(* PLC project Tc2_Utilities.PLC_ReadSymInfoByName Demo, tc3-libraries-kb TwinCAT 3.1 *)
(* stored: creationDateTime 2026-05-10T20:00:00, modificationDateTime 2026-05-10T20:00:00 *)

PROGRAM P_Demo_PLC_ReadSymInfoByName
  VAR
    fbPLC_ReadSymInfoByName : PLC_ReadSymInfoByName;  (* Tc2_Utilities.PLC_ReadSymInfoByName 实例 *)
    arg_NETID : T_AmsNetId;  (* VAR_INPUT NETID *)
    arg_PORT : T_AmsPort;  (* VAR_INPUT PORT *)
    arg_SYMNAME : T_MaxString;  (* VAR_INPUT SYMNAME *)
    arg_START : BOOL;  (* VAR_INPUT START *)
    arg_TMOUT : TIME;  (* VAR_INPUT TMOUT *)
    out_BUSY : BOOL;  (* VAR_OUTPUT BUSY *)
    out_ERR : BOOL;  (* VAR_OUTPUT ERR *)
    out_ERRID : UDINT;  (* VAR_OUTPUT ERRID *)
    out_SymInfo : SYMINFOSTRUCT;  (* VAR_OUTPUT SymInfo *)
  END_VAR

            // ============================================================
// Tc2_Utilities.PLC_ReadSymInfoByName 演示程序（FB 实例）
// ============================================================
// 验证步骤：
//   1. 引用 Tc2_Utilities（及依赖类型所在库 Tc2_System 等）
//   2. 编译 + 登录
//   3. 按 doc.md 给 arg_* 赋值
//   4. 在线监视 out_* / io_* 输出
// ============================================================

fbPLC_ReadSymInfoByName(
    NETID := arg_NETID,
    PORT := arg_PORT,
    SYMNAME := arg_SYMNAME,
    START := arg_START,
    TMOUT := arg_TMOUT,
    BUSY => out_BUSY,
    ERR => out_ERR,
    ERRID => out_ERRID,
    SymInfo => out_SymInfo
);

          
END_PROGRAM
